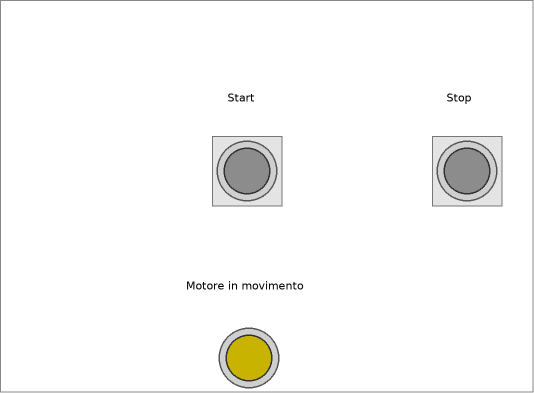
VISUALIZATION Visualization  // 534x393
    PushSwitch (212,136 70x70), variable: Gvl.PbStart, behaviour: TAP, style: Switch-PushSwitch-Gray
    PushSwitch (432,136 70x70), variable: Gvl.PbStop, behaviour: TAP, style: Switch-PushSwitch-Gray
    Label (166,83 150x30), "Start"
    Label (384,83 150x30), "Stop"
    Lamp1 (214,323 70x70), variable: Gvl.Axis.Status.Moving, style: Lamp-Lamp1-Yellow
    Label (170,271 150x30), "Motore in movimento"
END_VISUALIZATION

(* stored: Version 1.1.0.1, ProductVersion 3.1.4024.12
   Visu Visualization: Id {a42bbdd3-4374-4617-a748-c9c875916220} *)
